// TIA Portal V17 export
// export: Created 2023-12-22T15:04:40.3589601Z, ExportSetting WithDefaults, DisplayName Totally Integrated Automation Portal, DisplayVersion V17, DisplayName TIA Portal Openness, DisplayVersion V17, DisplayName TIA Portal Version Control Interface, DisplayVersion V17, DisplayName STEP 7 Professional, DisplayVersion V17, DisplayName STEP 7 Safety, DisplayVersion V17, DisplayName WinCC Advanced, DisplayVersion V17
FUNCTION_BLOCK "Slow"   // FB151, LAD
{ S7_Optimized_Access := 'FALSE' }
VERSION : 0.1
// stored: AutoNumber false, IsIECCheckEnabled false, SetENOAutomatically false, UDAEnableTagReadback false
   VAR_INPUT
      SP : Real;   // Уставка
   END_VAR
   VAR_IN_OUT
      Result : Real;   // Управляющий сигнал
   END_VAR
   VAR DB_SPECIFIC
      Use_Up { S7_SetPoint := 'True'} : Bool;   // Использовать плавный разгон
      Use_Down { S7_SetPoint := 'True'} : Bool;   // Использовать плавное замедление
      Active : Bool;   // Идёт изменение уставки
      Active_Up : Bool;
      Active_Down : Bool;
      Step_Up { S7_SetPoint := 'True'} : Real := 0.125;   // Шаг плавного разгона
      Step_Down { S7_SetPoint := 'True'} : Real := 0.125;   // Шаг плавного замедления
   END_VAR
   VAR
      T_Up { S7_SetPoint := 'True'} : "Time_R";   // Таймер плавного разгона
      T_Down { S7_SetPoint := 'True'} : "Time_R";   // Таймер плавного замедления
   END_VAR
   VAR_TEMP
      Delta_Up : Real;   // Отклонение сигнала от уставки
      Delta_Down : Real;
   END_VAR
   VAR_TEMP   // added for the SCL form of the ladder/FBD networks
      _w1 : Bool;
      _w2 : Bool;
   END_VAR
BEGIN

REGION Network 1: Не используется
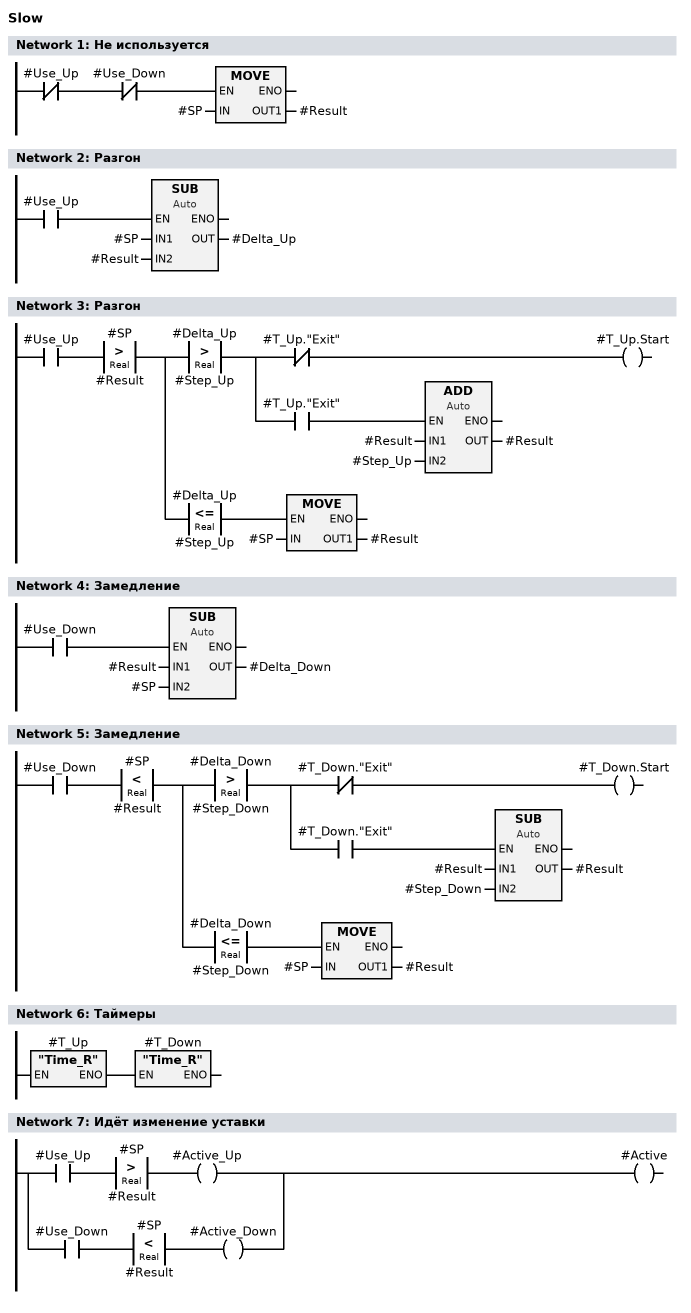
   RUNG wire#powerrail
      I_Contact( #Use_Up )
      I_Contact( #Use_Down )
      Move(in := #SP, out1 => #Result)
   END_RUNG
   // the same network as SCL:
   IF NOT #Use_Up AND NOT #Use_Down THEN #Result := #SP; END_IF;
END_REGION

REGION Network 2: Разгон
   RUNG wire#powerrail
      Contact( #Use_Up )
      Sub(in1 := #SP, in2 := #Result, out => #Delta_Up)
   END_RUNG
   // the same network as SCL:
   IF #Use_Up THEN #Delta_Up := #SP - #Result; END_IF;
END_REGION

REGION Network 3: Разгон
   RUNG wire#powerrail
      Contact( #Use_Up )
      { S7_Templates := "SrcType := Real" } GT_Contact(in1 := #SP, in2 := #Result)
      wire#w1
      { S7_Templates := "SrcType := Real" } GT_Contact(in1 := #Delta_Up, in2 := #Step_Up)
      wire#w2
      I_Contact( #T_Up."Exit" )
      Coil( #T_Up.Start )
   END_RUNG
   RUNG wire#w2
      Contact( #T_Up."Exit" )
      Add(in1 := #Result, in2 := #Step_Up, out => #Result)
   END_RUNG
   RUNG wire#w1
      { S7_Templates := "SrcType := Real" } LE_Contact(in1 := #Delta_Up, in2 := #Step_Up)
      Move(in := #SP, out1 => #Result)
   END_RUNG
   // the same network as SCL:
   #_w1 := #Use_Up AND (#SP > #Result);
   #_w2 := #_w1 AND (#Delta_Up > #Step_Up);
   #T_Up.Start := #_w2 AND NOT #T_Up."Exit";
   IF #_w2 AND #T_Up."Exit" THEN #Result := #Result + #Step_Up; END_IF;
   IF #_w1 AND (#Delta_Up <= #Step_Up) THEN #Result := #SP; END_IF;
END_REGION

REGION Network 4: Замедление
   RUNG wire#powerrail
      Contact( #Use_Down )
      Sub(in1 := #Result, in2 := #SP, out => #Delta_Down)
   END_RUNG
   // the same network as SCL:
   IF #Use_Down THEN #Delta_Down := #Result - #SP; END_IF;
END_REGION

REGION Network 5: Замедление
   RUNG wire#powerrail
      Contact( #Use_Down )
      { S7_Templates := "SrcType := Real" } LT_Contact(in1 := #SP, in2 := #Result)
      wire#w1
      { S7_Templates := "SrcType := Real" } GT_Contact(in1 := #Delta_Down, in2 := #Step_Down)
      wire#w2
      I_Contact( #T_Down."Exit" )
      Coil( #T_Down.Start )
   END_RUNG
   RUNG wire#w2
      Contact( #T_Down."Exit" )
      Sub(in1 := #Result, in2 := #Step_Down, out => #Result)
   END_RUNG
   RUNG wire#w1
      { S7_Templates := "SrcType := Real" } LE_Contact(in1 := #Delta_Down, in2 := #Step_Down)
      Move(in := #SP, out1 => #Result)
   END_RUNG
   // the same network as SCL:
   #_w1 := #Use_Down AND (#SP < #Result);
   #_w2 := #_w1 AND (#Delta_Down > #Step_Down);
   #T_Down.Start := #_w2 AND NOT #T_Down."Exit";
   IF #_w2 AND #T_Down."Exit" THEN #Result := #Result - #Step_Down; END_IF;
   IF #_w1 AND (#Delta_Down <= #Step_Down) THEN #Result := #SP; END_IF;
END_REGION

REGION Network 6: Таймеры
   RUNG wire#powerrail
      #T_Up()
      #T_Down()
   END_RUNG
   // the same network as SCL:
   #T_Up(ENO => #_w1);   // "Time_R"
   IF #_w1 THEN
       #T_Down();   // "Time_R"
   END_IF;
END_REGION

REGION Network 7: Идёт изменение уставки
   RUNG wire#powerrail
      Contact( #Use_Up )
      { S7_Templates := "SrcType := Real" } GT_Contact(in1 := #SP, in2 := #Result)
      Coil( #Active_Up )
      wire#w1
      Coil( #Active )
   END_RUNG
   RUNG wire#powerrail
      Contact( #Use_Down )
      { S7_Templates := "SrcType := Real" } LT_Contact(in1 := #SP, in2 := #Result)
      Coil( #Active_Down )
   END_RUNG wire#w1
   // the same network as SCL:
   #Active_Up := #Use_Up AND (#SP > #Result);
   #Active_Down := #Use_Down AND (#SP < #Result);
   #Active := #Active_Up OR #Active_Down;
END_REGION
END_FUNCTION_BLOCK
